(* CODESYS project raspberry_can.project

Project tree, tasks and I/O mapping:
  Device : CODESYS Control for Raspberry Pi SL, 3S - Smart Software Solutions GmbH, version 3.5.12.10
    application Application
      libraries: Standard, * (System); CAN API, 1.0.0.3 (3S - Smart Software Solutions GmbH); Util, * (System); VisuDialogs, * (System); BASIC, * (OSCAT); CAA Mathematics, 3.5.12.0 (CAA Technical Workgroup); CAA DTUtil Extern, 3.5.12.0 (CAA Technical Workgroup); CAA Real Time Clock Extern, 3.5.10.0 (CAA Technical Workgroup); SysTime, 3.5.9.0 (System)
      task MainTask (cyclic, interval t#20ms, priority 1) calls CAN_Master, Update_Visu
      task VISU_TASK (cyclic, interval 100 ms, priority 31) calls VisuElems.Visu_Prg
      global variables GVL
      function block MsgProcessor [ST]: ProcessMessage
      program CAN_Master [ST]
      visualisation Relative_Movement
      visualisation Visualization
      visualisation Absolute_Movement
      data type STATE
      data type CONVERT
      program Update_Visu [ST]
      function Math_Adjust [ST]
    Camera device
      <Empty>
    Onewire
    GPIOs_A_B : GPIOs A/B, 3S - Smart Software Solutions GmbH, version 3.5.11.0
        unmapped channels: digital inputs (GPIO0..GPIO31), digital outputs (GPIO0..GPIO31)
    SPI
    SoftMotion General Axis Pool
    I²C
  text list GlobalTextList
*)

// Device/Application/STATE
TYPE STATE :
(
	WAIT:= 0,   (* Wait for on button to be pressed*)
	INIT,       (*  Create messages *)
	SEND,		(* Send messages *)
	READ,		(* Receive messages *)
	PROCESS,    (* Process messages *)
	CANCEL      (* Cancel the creation of a message *)
);
END_TYPE

// Device/Application/CONVERT
TYPE CONVERT :
UNION
	myLReal: LREAL;
	myData: ARRAY [0..7] OF BYTE;
END_UNION
END_TYPE

// Device/Application/GVL
VAR_GLOBAL
	(* Message count *)
	g_countMsg_ST	: UINT;
	
	(* This data type descripes the configuration of the CANbus Driver *)
	g_busConfig		: CAN.DRIVER_CONFIG := (usiNetwork:= 0, uiBaudrate:= 500, ctMessages:= 10); 
	(* Time limit for receiving messages. T#0s:= no time limit *)
	g_tTimeLimit		: TIME := T#0s;
	home: BOOL;
	mode: INT;
	ok: BOOL;
	on: BOOL;
	cancel: BOOL;
	candle: BOOL;
	joint: ARRAY[1..6] OF REAL;
	initialPos: ARRAY[1..6] OF REAL;
	currentPos: ARRAY[1..6] OF REAL;
	// 0 indicates radians and 1 indicates degrees
	anglesMode: BOOL;
	error: ARRAY[1..6] OF REAL;
	desiredPos: ARRAY[1..6] OF REAL;
END_VAR

// Device/Application/CAN_Master
PROGRAM CAN_Master
VAR	
	// State of the program
	eSTATE: STATE;
	uCONVERT: CONVERT;
	(* A CANbus for handling 11bit CobIds *)
	driver11bit		: CAN.CANBus_11bit := ( DriverConfig:= g_busConfig );

	(* Handle for an Mask Receiver *)
	hMaskReceiver	: CAN.CAA.HANDLE;
			
	(* Received messages are passed to MessageProcessors. *)
	msgProcessor	: MsgProcessor;
	
	(* Defines a mask for the receiver *)
	maskConfig		: CAN.RECEIVER_MASK := (
										dwIdValue:= 0, 
										dwIdMask:= 0, 
										xRTRValue:= FALSE, 
										xRTRMask:= FALSE, 
										x29BitIdValue:= FALSE, 
										x29BitIdMask:= FALSE, 
										xTransmitValue:= FALSE, 
										xTransmitMask:= TRUE, 
										xAlwaysNewest:= FALSE);
	(* The messages received by the receiver *)
	msgSend	: ARRAY[0..6] OF CAN.RxMESSAGE;
	i: INT;
	j: INT;
	_pdriver11bit: POINTER TO CAN.CANBus_11bit;
END_VAR

CASE eSTATE OF
	
STATE.WAIT:  // wait for button on to be pressed
	IF on THEN 
		eSTATE:= STATE.INIT;
	END_IF


STATE.INIT:
	// Configure CAN Driver
	driver11bit(DriverConfig:= g_busConfig, eError=> );
	_pdriver11bit := ADR(driver11bit);
	
	// Define frame's properties
	FOR i:= 0 TO 6 DO
		msgSend[i].usiDataLength:= 8;
		msgSend[i].udiCanID:= 123;
		msgSend[i].xRTR:= 0;
		msgSend[i].xIs29BitMessage:= 0;
	END_FOR
	
	// Create 7 messages
	IF NOT(GVL.home) AND NOT(GVL.candle) THEN
		
		// Create first message carrying the mode selected
		IF GVL.mode = 1 THEN
			uCONVERT.myLReal:= 1.0;
		ELSIF GVL.mode = 0 THEN  
			uCONVERT.myLReal:= 0.0;
		END_IF
		
		FOR j:= 0 TO 7 DO
			msgSend[0].abyData[j]:= uCONVERT.myData[j];
		END_FOR
	
		// Create 6 next messages carrying the desired joint positions
		FOR i:= 1 TO 6 DO 
			uCONVERT.myLReal:= OSCAT_BASIC.ROUND(GVL.joint[i], 2);	
			FOR j:= 0 TO 7 DO
				msgSend[i].abyData[j]:= uCONVERT.myData[j];
			END_FOR
		END_FOR		
		
	ELSIF GVL.home THEN
	 	uCONVERT.myLReal:= 0.0;
		FOR j:= 0 TO 7 DO
			msgSend[0].abyData[j]:= uCONVERT.myData[j];
			msgSend[1].abyData[j]:= uCONVERT.myData[j];
			msgSend[6].abyData[j]:= uCONVERT.myData[j];
		END_FOR
		
		uCONVERT.myLReal:= 2.9;	
		FOR j:= 0 TO 7 DO
			msgSend[2].abyData[j]:= uCONVERT.myData[j];
		END_FOR
		
		uCONVERT.myLReal:= 1.3;	
		FOR j:= 0 TO 7 DO
			msgSend[3].abyData[j]:= uCONVERT.myData[j];
		END_FOR
		
		uCONVERT.myLReal:= 4.2;	
		FOR j:= 0 TO 7 DO
			msgSend[4].abyData[j]:= uCONVERT.myData[j];
		END_FOR
		
		uCONVERT.myLReal:= 1.4;	
		FOR j:= 0 TO 7 DO
			msgSend[5].abyData[j]:= uCONVERT.myData[j];
		END_FOR
		
	ELSIF GVL.candle THEN 
		uCONVERT.myLReal:= 0.0;
		FOR j:= 0 TO 7 DO
			msgSend[0].abyData[j]:= uCONVERT.myData[j];
		END_FOR
	
		uCONVERT.myLReal:= 3.14;	
		FOR i:= 1 TO 6 DO 
			FOR j:= 0 TO 7 DO
				msgSend[i].abyData[j]:= uCONVERT.myData[j];
			END_FOR
		END_FOR
			
	END_IF
	
    IF GVL.cancel THEN
		eSTATE:= STATE.CANCEL; // recreate the message if button cancel is pressed
	ELSIF GVL.ok THEN
		eSTATE:= STATE.SEND;  // send message if button on is pressed
	END_IF
	
	
STATE.SEND:		
	// Send messages
	IF _pdriver11bit <> 0 AND ok THEN
		FOR i:= 0 TO 6 DO 
			_pdriver11bit^.SendMessage(Message:= msgSend[i], eError=> );
		END_FOR	
	END_IF
	
	GVL.ok:= 0;
	eState:= STATE.READ;
	
				
STATE.READ:
	// Configure MessageProcessor
	msgProcessor(CANdriver:= driver11bit);

	// Create a Mask Receiver to receive all messages
	IF hMaskReceiver = CAN.CAA.gc_hINVALID THEN
		hMaskReceiver:= driver11bit.GetMaskReceiver(Mask:= maskConfig, eError=> );
	END_IF
	// Receive messages and hand them over to the MsgProccessor
	driver11bit.ReceiveMessage(hReceiver:= hMaskReceiver, itfMsgProcessor:= msgProcessor, tTimeLimit:= g_tTimeLimit, eError=> );

	IF 	GVL.g_countMsg_ST = 6 THEN
		GVL.g_countMsg_ST:= 0;
		eSTATE:= STATE.PROCESS;
	END_IF
		

STATE.PROCESS:
	// Compute desired joint position	
	IF GVL.home THEN
		GVL.desiredPos[1]:= 0.0;
		GVL.desiredPos[2]:= 2.9;
		GVL.desiredPos[3]:= 1.3;
		GVL.desiredPos[4]:= 4.2;
		GVL.desiredPos[5]:= 1.4;
		GVL.desiredPos[6]:= 0.0;
		GVL.home:= 0;
	ELSIF GVL.candle THEN 
		FOR i:= 1 TO 6 DO
			GVL.desiredPos[i]:= 3.14;
		END_FOR
		GVL.candle:=0;
	ELSE
		FOR i:= 1 TO 6 DO
			GVL.desiredPos[i]:= GVL.initialPos[i] + GVL.joint[i];
		END_FOR
	END_IF

	// Compute position error
	FOR i:= 1 TO 6 DO
		GVL.error[i]:= Math_Adjust(Math_Adjust(GVL.desiredPos[i]) - Math_Adjust(GVL.currentPos[i]));
		GVL.error[i]:= OSCAT_BASIC.ROUND(in:= error[i], N:= 6);
	END_FOR

	// Set initial joint position for the next execution 
	FOR i:= 1 TO 6 DO
		GVL.initialPos[i]:= OSCAT_BASIC.ROUND(in:= GVL.currentPos[i], N:= 6);
	END_FOR	
	
	eSTATE:= STATE.INIT;


STATE.CANCEL:
	GVL.home:= 0;
	GVL.candle:= 0;
	GVL.cancel:= 0;
	eSTATE:= STATE.INIT;
		
END_CASE

END_PROGRAM

// Device/Application/MsgProcessor
// MsgProcessor is the implimentation of IMessageProcessor
FUNCTION_BLOCK MsgProcessor IMPLEMENTS CAN.IMessageProcessor
VAR_IN_OUT
	CANdriver	: CAN.CANBus_11bit;
END_VAR

VAR
	_pCANdriver : POINTER TO CAN.CANBus_11bit;
END_VAR

_pCANdriver := ADR(CANdriver);

METHOD ProcessMessage
VAR_IN_OUT
	(* The messages received by the receiver *)
	Message	: CAN.RxMessage;
END_VAR
VAR
	i: INT;
	unCONVERT: CONVERT;
END_VAR
// Retrieve current state from received message
g_countMsg_ST:= g_countMsg_ST +1;  // count received messages

FOR i:= 0 TO 7 DO
	unCONVERT.myData[i]:= Message.abyData[i];
END_FOR

GVL.currentPos[GVL.g_countMsg_ST]:= LREAL_TO_REAL(unCONVERT.myLReal);
END_METHOD

END_FUNCTION_BLOCK

// Device/Application/Math_Adjust
// Function that computes the angular position error of each joint within the
// range of 0 to 2pi rad.
FUNCTION Math_Adjust : REAL
VAR_INPUT
	value: REAL;
END_VAR

IF value <= -3.14 OR value > 3.14 THEN
	Math_adjust:= LREAL_TO_REAL(MATH.fmod(lrX:= value, lrM:= 6.28));
	IF value <= -3.14 THEN 
		Math_adjust:= value + 6.28;
	ELSIF value > 3.14 THEN
		Math_adjust:= value - 6.28;
	END_IF
ELSE
	Math_adjust:= value;
END_IF

END_FUNCTION

// Device/Application/Update_Visu
// Program responsible to update visualization textfields, buttons etc.
// regarding with the user's choices.
PROGRAM Update_Visu
VAR
	joint2MinStr: STRING;
	joint2MaxStr: STRING;
	joint3MinStr: STRING;
	joint3MaxStr: STRING;
	joint2Min: REAL;
	joint2Max: REAL;
	joint3Min: REAL;
	joint3Max: REAL;
	constraintsMin: ARRAY[1..6] OF REAL := [-3.14, 0.87, 0.33, -3.14, -3.14, -3.14];
	constraintsMax: ARRAY[1..6] OF REAL := [3.14, 5.41, 5.95, 3.14, 3.14, 3.14];
	anglesModeStr: STRING;
	jointVisu: ARRAY [1..6] OF STRING;
	errorVisu: ARRAY [1..6] OF STRING;
	currentPosVisu: ARRAY [1..6] OF STRING;
	constraintsMinVisu: ARRAY [1..6] OF STRING;
	constraintsMaxVisu: ARRAY [1..6] OF STRING;
	alarm: BOOL;
	alarm1: BOOL;
	alarm4: BOOL;
	alarm5: BOOL;
	alarm6: BOOL;
	i: INT;
END_VAR

// Update visualization elements according to user's choices
joint2Min:= OSCAT_BASIC.ROUND(constraintsMin[2] - GVL.initialPos[2], 2);
joint2Max:= OSCAT_BASIC.ROUND(constraintsMax[2] - GVL.initialPos[2], 2);
joint3Min:= OSCAT_BASIC.ROUND(constraintsMin[3] - GVL.initialPos[3], 2);
joint3Max:= OSCAT_BASIC.ROUND(constraintsMax[3] - GVL.initialPos[3], 2);

IF GVL.anglesMode = 0 THEN
	
	anglesModeStr:= 'DEG';
	
	FOR i:= 1 TO 6 DO
		jointVisu[i]:= REAL_TO_STRING(OSCAT_BASIC.ROUND(GVL.joint[i], 2));
		constraintsMinVisu[i]:= REAL_TO_STRING(constraintsMin[i]);
		constraintsMaxVisu[i]:= REAL_TO_STRING(constraintsMax[i]);
		currentPosVisu[i]:= REAL_TO_STRING(OSCAT_BASIC.ROUND(GVL.currentPos[i], 6));
		errorVisu[i]:= REAL_TO_STRING(OSCAT_BASIC.ROUND(GVL.error[i], 6));
	END_FOR
	
	joint2MinStr:= REAL_TO_STRING(joint2Min);
	joint2MaxStr:= REAL_TO_STRING(joint2Max);
	joint3MinStr:= REAL_TO_STRING(joint3Min);
	joint3MaxStr:= REAL_TO_STRING(joint3Max);
	
ELSIF GVL.anglesMode = 1 THEN
	
	anglesModeStr:= 'RAD';
	
	FOR i:= 1 TO 6 DO
		jointVisu[i]:= INT_TO_STRING(REAL_TO_INT(OSCAT_BASIC.ROUND(GVL.joint[i] / 3.14 * 180, 0)));
		constraintsMinVisu[i]:= INT_TO_STRING(REAL_TO_INT(OSCAT_BASIC.ROUND(constraintsMin[i] / 3.14 * 180, 0 )));
		constraintsMaxVisu[i]:= INT_TO_STRING(REAL_TO_INT(OSCAT_BASIC.ROUND(constraintsMax[i] / 3.14 * 180, 0)));
		currentPosVisu[i]:= INT_TO_STRING(REAL_TO_INT(OSCAT_BASIC.ROUND(GVL.currentPos[i] / 3.14 * 180, 2)));
		errorVisu[i]:= INT_TO_STRING(REAL_TO_INT(OSCAT_BASIC.ROUND(GVL.error[i] / 3.14 * 180, 2)));
	END_FOR
	
	joint2MinStr:= INT_TO_STRING(REAL_TO_INT(OSCAT_BASIC.ROUND(joint2Min / 3.14 * 180, 0)));
	joint2MaxStr:= INT_TO_STRING(REAL_TO_INT(OSCAT_BASIC.ROUND(joint2Max / 3.14 * 180, 0)));
	joint3MinStr:= INT_TO_STRING(REAL_TO_INT(OSCAT_BASIC.ROUND(joint3Min / 3.14 * 180, 0)));
	joint3MaxStr:= INT_TO_STRING(REAL_TO_INT(OSCAT_BASIC.ROUND(joint3max / 3.14 * 180, 0)));
		
END_IF

// Check if joints 1, 4, 5, 6 are about to reach 10000 degrees or -10000 degrees
IF GVL.currentPos[1] / 3.14 * 180 >= 9280 OR GVL.currentPos[1] / 3.14 * 180 <= -9280 THEN
	alarm1:= 1;
	alarm:= 1;
ELSIF GVL.currentPos[4] / 3.14 * 180 >= 9280 OR GVL.currentPos[4] / 3.14 * 180 <= -9280 THEN
	alarm4:= 1;
	alarm:= 1;
ELSIF GVL.currentPos[5] / 3.14 * 180 >= 9280 OR GVL.currentPos[5] / 3.14 * 180 <= -9280 THEN
	alarm5:= 1;
	alarm:= 1;
ELSIF GVL.currentPos[6] / 3.14 * 180 >= 9280 OR GVL.currentPos[6] / 3.14 * 180 <= -9280 THEN
	alarm6:= 1;
	alarm:= 1;
ELSE
	alarm1:= 0;
	alarm4:= 0;
	alarm5:= 0;
	alarm6:= 0;
	alarm:= 0;
END_IF

END_PROGRAM

// Device/Application/Relative_Movement
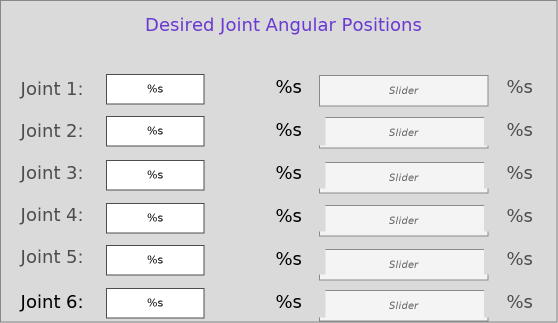
VISUALIZATION Relative_Movement  // 558x323
    Slider (319,117 169x31), variable: GVL.joint[2], scale 0.87..5.41
    Slider (319,162 169x31), variable: GVL.joint[3], scale 0.33..5.95
    Slider (319,205 169x31), variable: GVL.joint[4], scale -3.14..3.14
    Slider (319,249 169x31), variable: GVL.joint[5], scale -3.14..3.14
    Slider (319,290 169x31), variable: GVL.joint[6], scale -3.14..3.14
    Label (111,10 345x30), "Desired Joint Angular Positions"
    Textfield (106,74 98x30), "%s", text variable: Update_Visu.jointVisu[1]
        OnMouseClick: write joint[1] via Edit
    Textfield (106,116 98x30), "%s", text variable: Update_Visu.jointVisu[2]
        OnMouseClick: write joint[2] via Edit
    Textfield (106,160 98x30), "%s", text variable: Update_Visu.jointVisu[3]
        OnMouseClick: write joint[3] via Edit
    Textfield (106,203 98x30), "%s", text variable: Update_Visu.jointVisu[4]
        OnMouseClick: write joint[4] via Edit
    Textfield (106,245 98x30), "%s", text variable: Update_Visu.jointVisu[5]
        OnMouseClick: write joint[5] via Edit
    Textfield (106,288 98x30), "%s", text variable: Update_Visu.jointVisu[6]
        OnMouseClick: write joint[6] via Edit
    Label (14,70 76x38), "Joint 1:"
    Label (14,112 76x38), "Joint 2:"
    Label (14,154 76x38), "Joint 3:"
    Label (14,196 76x38), "Joint 4:"
    Label (14,238 76x38), "Joint 5:"
    Label (14,283 76x38), "Joint 6:"
    Textfield (484,72 72x30), "%s", text variable: Update_Visu.constraintsMaxVisu[1]
    Textfield (484,115 72x30), "%s", text variable: Update_Visu.joint2MaxStr
    Textfield (484,158 72x30), "%s", text variable: Update_Visu.joint3MaxStr
    Textfield (484,201 72x30), "%s", text variable: Update_Visu.constraintsMaxVisu[4]
    Textfield (484,244 72x30), "%s", text variable: Update_Visu.constraintsMaxVisu[5]
    Textfield (484,287 72x30), "%s", text variable: Update_Visu.constraintsMaxVisu[6]
    Textfield (253,72 72x30), "%s", text variable: Update_Visu.constraintsMinVisu[1]
    Textfield (253,115 72x30), "%s", text variable: Update_Visu.joint2MinStr
    Textfield (253,158 72x30), "%s", text variable: Update_Visu.joint3MinStr
    Textfield (253,201 72x30), "%s", text variable: Update_Visu.constraintsMinVisu[4]
    Textfield (253,244 72x30), "%s", text variable: Update_Visu.constraintsMinVisu[5]
    Textfield (253,287 72x30), "%s", text variable: Update_Visu.constraintsMinVisu[6]
    Slider (319,75 169x31), variable: GVL.joint[1], scale -3.14..3.14
END_VISUALIZATION

// Device/Application/Visualization
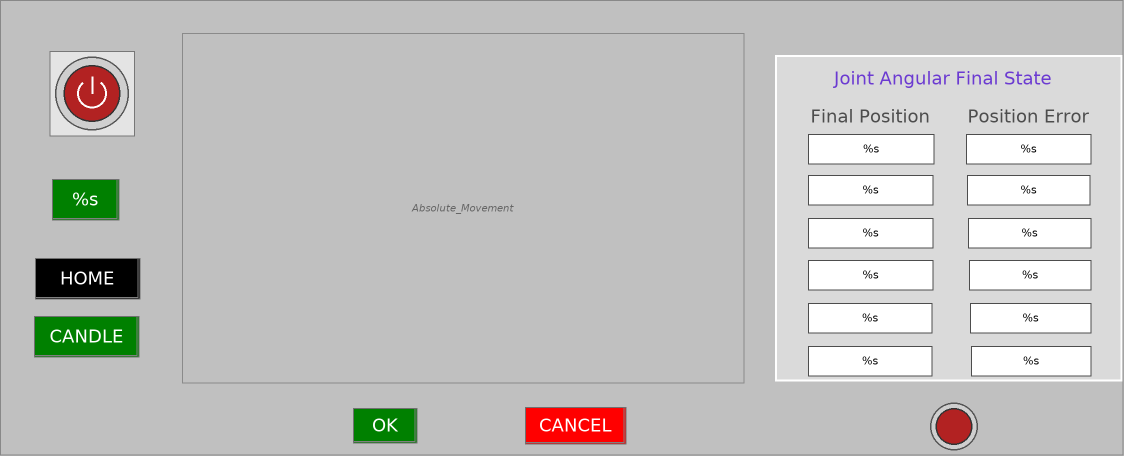
VISUALIZATION Visualization  // 1124x456
    Rectangle (775,55 347x326)
    PowerSwitch (47,51 90x85), variable: GVL.on, behaviour: TOGGLE, style: Switch-PowerSwitch-Red
    Textfield (808,134 126x30), "%s", text variable: Update_Visu.currentPosVisu[1], colour toggle: Update_Visu.alarm1
        p2167032090: 16#FF0000
    Textfield (808,175 125x30), "%s", text variable: Update_Visu.currentPosVisu[2]
    Textfield (808,218 125x30), "%s", text variable: Update_Visu.currentPosVisu[3]
    Textfield (808,260 125x30), "%s", text variable: Update_Visu.currentPosVisu[4], colour toggle: Update_Visu.alarm4
        p3092690914: 16#FF0000
    Textfield (808,303 124x30), "%s", text variable: Update_Visu.currentPosVisu[5], colour toggle: Update_Visu.alarm5
        p3092690914: 16#FF0000
    Textfield (808,346 124x30), "%s", text variable: Update_Visu.currentPosVisu[6], colour toggle: Update_Visu.alarm6
        p3092690914: 16#FF0000
    Label (800,100 141x33), "Final Position"
    TabControl (182,33 562x350), input disabled if: not (GVL.on), frame switch variable: GVL.mode
        shows Absolute_Movement()
        shows Relative_Movement()
        [0]: TabTitle=Absolute Movement
        [1]: TabTitle=Relative Movement
    Button (35,258 105x41), "HOME", input disabled if: not (GVL.on)
        toggle GVL.home
    Button (34,316 105x41), "CANDLE", input disabled if: not (GVL.on)
        toggle GVL.candle
    Label (797,66 292x25), "Joint Angular Final State"
    Textfield (966,134 125x30), "%s", text variable: Update_Visu.errorVisu[1]
    Textfield (967,175 123x30), "%s", text variable: Update_Visu.errorVisu[2]
    Textfield (968,218 123x30), "%s", text variable: Update_Visu.errorVisu[3]
    Textfield (969,260 122x30), "%s", text variable: Update_Visu.errorVisu[4]
    Textfield (970,303 121x30), "%s", text variable: Update_Visu.errorVisu[5]
    Textfield (971,346 120x30), "%s", text variable: Update_Visu.errorVisu[6]
    Label (959,100 139x33), "Position Error"
    Button (353,408 64x35), "OK", input disabled if: not (GVL.on)
        toggle GVL.ok
    Button (525,407 101x37), "CANCEL", input disabled if: not (GVL.on)
        toggle GVL.cancel
    Button (52,179 67x41), "%s", text variable: Update_Visu.anglesModeStr, input disabled if: not (GVL.on)
        toggle GVL.anglesMode
    Lamp1 (926,399 56x55), variable: Update_Visu.alarm, style: Lamp-Lamp1-Red
END_VISUALIZATION

// Device/Application/Absolute_Movement
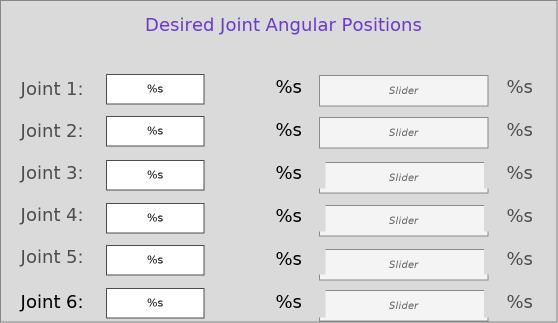
VISUALIZATION Absolute_Movement  // 558x323
    Slider (319,162 169x31), variable: GVL.joint[3], scale 0.33..5.95
    Slider (319,205 169x31), variable: GVL.joint[4], scale -3.14..3.14
    Slider (319,249 169x31), variable: GVL.joint[5], scale -3.14..3.14
    Slider (319,290 169x31), variable: GVL.joint[6], scale -3.14..3.14
    Label (111,10 345x30), "Desired Joint Angular Positions"
    Textfield (106,74 98x30), "%s", text variable: Update_Visu.jointVisu[1]
        OnMouseClick: write joint[1] via Edit
    Textfield (106,116 98x30), "%s", text variable: Update_Visu.jointVisu[2]
        OnMouseClick: write joint[2] via Edit
    Textfield (106,160 98x30), "%s", text variable: Update_Visu.jointVisu[3]
        OnMouseClick: write joint[3] via Edit
    Textfield (106,203 98x30), "%s", text variable: Update_Visu.jointVisu[4]
        OnMouseClick: write joint[4] via Edit
    Textfield (106,245 98x30), "%s", text variable: Update_Visu.jointVisu[5]
        OnMouseClick: write joint[5] via Edit
    Textfield (106,288 98x30), "%s", text variable: Update_Visu.jointVisu[6]
        OnMouseClick: write joint[6] via Edit
    Label (14,70 76x38), "Joint 1:"
    Label (14,112 76x38), "Joint 2:"
    Label (14,154 76x38), "Joint 3:"
    Label (14,196 76x38), "Joint 4:"
    Label (14,238 76x38), "Joint 5:"
    Label (14,283 76x38), "Joint 6:"
    Textfield (484,72 72x30), "%s", text variable: Update_Visu.constraintsMaxVisu[1]
    Textfield (484,115 72x30), "%s", text variable: Update_Visu.constraintsMaxVisu[2]
    Textfield (484,158 72x30), "%s", text variable: Update_Visu.constraintsMaxVisu[3]
    Textfield (484,201 72x30), "%s", text variable: Update_Visu.constraintsMaxVisu[4]
    Textfield (484,244 72x30), "%s", text variable: Update_Visu.constraintsMaxVisu[5]
    Textfield (484,287 72x30), "%s", text variable: Update_Visu.constraintsMaxVisu[6]
    Textfield (253,72 72x30), "%s", text variable: Update_Visu.constraintsMinVisu[1]
    Textfield (253,115 72x30), "%s", text variable: Update_Visu.constraintsMinVisu[2]
    Textfield (253,158 72x30), "%s", text variable: Update_Visu.constraintsMinVisu[3]
    Textfield (253,201 72x30), "%s", text variable: Update_Visu.constraintsMinVisu[4]
    Textfield (253,244 72x30), "%s", text variable: Update_Visu.constraintsMinVisu[5]
    Textfield (253,287 72x30), "%s", text variable: Update_Visu.constraintsMinVisu[6]
    Slider (319,75 169x31), variable: GVL.joint[1], scale -3.14..3.14
    Slider (319,117 169x31), variable: GVL.joint[2], scale 0.87..5.41
END_VISUALIZATION
